FUNCTION_BLOCK Stamp EXTENDS BaseComponent
VAR_INPUT
END_VAR
VAR_OUTPUT
END_VAR
VAR
	m_stampingCylinder: MonostableCylinder;
	m_slidingCylinder: BistableCylinder;
	m_pressureValve: PropotionalValve;
	
	m_presenceSensor: PresenceSensor;
	m_pressureSensor: PressureSensor;
END_VAR

PROPERTY StampPressure : INT
GET
StampPressure:=m_pressureSensor.Value;
END_GET
SET
m_pressureValve.Pressure := StampPressure;
END_SET
END_PROPERTY

PROPERTY WPAtStart : BOOL
GET
WPAtStart := m_presenceSensor.Value;
END_GET
END_PROPERTY

END_FUNCTION_BLOCK

(* stored: Version 1.1.0.1
   POU Stamp: Id {1f493665-2321-4012-b50d-e272b9c0b026}, SpecialFunc None
   Property StampPressure: Id {9b39b37f-8ddd-4fa6-9a41-5d43fec26aa9}
   Get Get: Id {aad7feae-229d-433d-8039-98c7ef4b7198}
   Set Set: Id {32608fd9-633f-4f17-922d-d80f1d26becf}
   Property WPAtStart: Id {af469093-14af-413b-8ce5-d86c657b748f}
   Get Get: Id {7599df50-edc3-483d-980c-ec41d4dc7332} *)
